FUNCTION_BLOCK FB_MollineC3HeatCounter
VAR_INPUT
	aHeatCounterTelegramm : ARRAY[1..cMBUS_MaxTelegrams] OF ST_MBus_Data2;
END_VAR
VAR_OUTPUT
	fFeedTemperature : REAL; //°C
	fReturnTemperazure : REAL; //°C
	fVolumeFlowRate : REAL; //m3/s
END_VAR
VAR
	{attribute 'OPC.UA.DA' := '1'}
	sensorState : ST_MollineC3HeatCounterState;
END_VAR

//set sensor state
sensorState.fVolume := STRING_TO_REAL(aHeatCounterTelegramm[1].arrData[3].sValue);
sensorState.fFeedTemperature := STRING_TO_REAL(aHeatCounterTelegramm[1].arrData[8].sValue);
sensorState.fReturnTemperature := STRING_TO_REAL(aHeatCounterTelegramm[1].arrData[9].sValue);
sensorState.fVolumeFlowRate := STRING_TO_REAL(aHeatCounterTelegramm[1].arrData[6].sValue);
sensorState.fHeatEnergy := STRING_TO_REAL(aHeatCounterTelegramm[1].arrData[2].sValue)/1000000;
sensorState.fTemperatureDifference := STRING_TO_REAL(aHeatCounterTelegramm[1].arrData[10].sValue);

//calculate fHeatFlowRate because heat meter does not measure negative flows
sensorState.fHeatFlowRate := sensorState.fVolumeFlowRate/3.6*4.19*sensorState.fTemperatureDifference;

//set outputs
fFeedTemperature := sensorState.fFeedTemperature;
fReturnTemperazure := sensorState.fReturnTemperature;
fVolumeFlowRate := sensorState.fVolumeFlowRate;

END_FUNCTION_BLOCK

(* stored: Version 1.1.0.1, ProductVersion 3.1.4024.10
   POU FB_MollineC3HeatCounter: Id {68b26994-e772-43d9-bb19-4685b29f39a6}, SpecialFunc None *)
